(* IEC 61131-3 sources: test/Class/_AccContMain (part 2) *)

        else
          SetMSGNr(dMSGNumber:=ERR_AUTHORITY_EDITUSER);
        end_if;

      else
        SetMSGNr(dMSGNumber:=ERR_USER_NOTEXIST);
      end_if;

    else
      SetMSGNr(dMSGNumber:=ERR_NO_NAME);
    end_if;

  else
    SetMSGNr(dMSGNumber:=ERR_DELUSER);
  end_if;

END_FUNCTION

FUNCTION GLOBAL _AccContMain::ShowUserData
  VAR
    tmpPos    : DINT;
    tmpUser   : t_s_UserV2;  //V2.29, dacpat, updated to new struct
  END_VAR

  tmpPos := -1;

  // Benutzername angegeben
  //-----------------------------------------------------------------------------------------
  if (StrEditUserName.GetLength()) then

      // Position des Benutzers holen
      //-----------------------------------------------------------------------------------------
      tmpPos := SearchUser(pBuffer := UsersBuffer, pUserName:=StrEditUserName.DataBuffer.GetDataPtr(), pUser:=#tmpUser);
      if (tmpPos >= 0) then

        // Benutzerdaten kopieren
        StrEditUserName.WriteDataOff(udLen:=_strlen(#tmpUser.aUsername[0]), udOff:=0, pData:=#tmpUser.aUsername[0]);
        StrEditPasswordOld.WriteDataOff(udLen:=1, udOff:=0, pData:="");
        StrEditPassword.WriteDataOff(udLen:=1, udOff:=0, pData:="");
        StrEditPassword2.WriteDataOff(udLen:=1, udOff:=0, pData:="");
        StrEditInfo.WriteDataOff(udLen:=_strlen(#tmpUser.aUserInfo[0]), udOff:=0, pData:=#tmpUser.aUserInfo[0]);
        ELevel   := tmpUser.usUserLevel;
        ETimeOut := tmpUser.udUserTimeout;

      else

        // Leere Daten kopieren
        StrEditUserName.WriteDataOff(udLen:=1, udOff:=0, pData:="");
        StrEditPasswordOld.WriteDataOff(udLen:=1, udOff:=0, pData:="");
        StrEditPassword.WriteDataOff(udLen:=1, udOff:=0, pData:="");
        StrEditPassword2.WriteDataOff(udLen:=1, udOff:=0, pData:="");
        StrEditInfo.WriteDataOff(udLen:=1, udOff:=0, pData:="");
        ELevel   := 0;
        ETimeOut := 0;

        SetMSGNr(dMSGNumber:=ERR_USER_NOTEXIST);

      end_if;

  else

    SetMSGNr(dMSGNumber:=ERR_NO_NAME);

  end_if;

END_FUNCTION

FUNCTION GLOBAL _AccContMain::ChangePassword
	VAR_INPUT
		bAdmin 	: BOOL;
	END_VAR
	VAR_OUTPUT
		bRet 	: BOOL;
	END_VAR
  VAR
  	tmpUserName   : ARRAY[0..AccessControl_MaxUsernameLength] of CHAR;
    tmpPassword   : ARRAY[0..AccessControl_MaxPasswordLength] of CHAR;
    tmpPWControl  : ARRAY[0..AccessControl_MaxPasswordLength] of CHAR;
    tmpUser       : t_s_UserV2;  //V2.29, dacpat, updated to new struct
    pActUser      : ^t_s_UserV2;  //V2.29, dacpat, updated to new struct
    tmpPos        : DINT;
    tmpPW1Length  : UDINT;
    tmpPW2Length  : UDINT;
  END_VAR

  bRet            := false;
  tmpUserName[0]  := 0;
  tmpPassword[0]  := 0;
  tmpPWControl[0] := 0;
  pActUser        := NIL;
  tmpPos          := 0;

  // Benutzer eingeloggt oder Benutzerverwaltung
  //-----------------------------------------------------------------------------------------
  if ((UserIsLoggedIn = true) | (bAdmin = true)) then

    // Benutzername und Passwörter holen
    if (bAdmin = true) then
      StrEditUserName.GetDataAt(pData:=#tmpUserName[0], udSize:=StrEditUserName.GetLength()+1, udAt:=0);
    else
      StrActUser.GetDataAt(pData:=#tmpUserName[0], udSize:=StrActUser.GetLength()+1, udAt:=0);
    end_if;
    tmpPW1Length := StrEditPassword.GetLength()+1;
    tmpPW2Length := StrEditPassword2.GetLength()+1;
    StrEditPassword.GetDataAt(pData:=#tmpPassword[0], udSize:=tmpPW1Length, udAt:=0);
    StrEditPassword2.GetDataAt(pData:=#tmpPWControl[0], udSize:=tmpPW2Length, udAt:=0);

    // Soll das PW geändert werden?
    //-----------------------------------------------------------------------------------------
    if ((tmpPW1Length > 1) & (tmpPW2Length > 1)) then

      // Geändertes Passwort richtig eingegeben?
      //-----------------------------------------------------------------------------------------
      if (StrCmp(p0:=#tmpPassword[0], x1:=sizeof(tmpPassword[0]), p2:=#tmpPWControl[0], x3:=sizeof(tmpPWControl[0])) = 0) then

        // Position des Benutzers holen
        tmpPos := SearchUser(pBuffer := UsersBuffer, pUserName:= #tmpUserName[0], pUser:=#tmpUser);
        if (tmpPos >= 0) then

          // Benutzerdaten anhand der Position holen und neues Passwort setzen
          //-----------------------------------------------------------------------------------------
          pActUser := getUserToEdit(udPos:=to_udint(tmpPos));
          if (pActUser <> NIL) then

            StrNCpy(p0 := #pActUser^.aUserPassword[0],
                    x1 := sizeof(pActUser^.aUserPassword[0]),
                    p2 := #tmpPassword[0],
                    x3 := sizeof(tmpPassword[0]),
                    ml := AccessControl_MaxPasswordLength);
            if (bAdmin = false) then
              refreshUserFile();
            end_if;
            SetMSGNr(dMSGNumber:=MSG_PWCHANGE_OK);
            bRet := true;

          end_if;

        else

          SetMSGNr(dMSGNumber:=ERR_USER_NOTEXIST);

        end_if;

      else

        SetMSGNr(dMSGNumber:=ERR_WRONG_PWCHANGE);

      end_if;

    else

      // Passwort nicht geändert
      bRet := FALSE;

    end_if;

  end_if;

END_FUNCTION

FUNCTION VIRTUAL GLOBAL _AccContMain::SelectFunction::Write
	VAR_INPUT
		input (EAX) 	: DINT;
	END_VAR
	VAR_OUTPUT
		result (EAX) 	: DINT;
	END_VAR

	SelectFunction := input;

  //*****************************************************************************
  //** Jeweilige Funktion ausgewählt                                           **
  //*****************************************************************************
  case SelectFunction of

    // Legt einen neuen Benutzer an
    1:  AddUser();
        clearServers();

    // Löscht den ausgewählten Benutzer
    2:  DeleteUser();
        clearServers();

    // Bearbeitet den ausgewählten Benutzer
    3:  EditUser();
        clearServers();

    // Login
    4:  Login();
        clearServers();

    // Logout
    5:  Logout();
        clearServers();

    // Schreibt die Benutzerdaten des ausgewählten Benutzers auf die Server zum Bearbeiten
    6:  ShowUserData();

    // Ändert das Passwort des ausgewählten Benutzers
    7:  ChangePassword(bAdmin:=false);
        clearServers();

    // Verknüpft die Seriennummer des aktuellen Speichermediums mit dem eingeloggten Benutzer
    8:  AddUsbSN();
        clearServers();

    // Verknüpft die Seriennummer des aktuellen Speichermediums mit dem eingeloggten Benutzer
    9:  AddUsbSNbyUser();
        clearServers();

    // Löscht die Verknüpfung der Seriennummer mit dem aktuellen Speichermedium
    10: DelUsbSN();
        clearServers();

    // Löscht alle Benutzerdaten auf den Servern
    11: clearServers();

    // Springt auf den vorherigen Bildschirm
    12: closeScreen();

    // V2.30, dacpat, RFID Login
    13:  IsRFIDUser := TRUE;
         Login();
         clearServers();

    // V2.30, dacpat, RFID Add User
    14:  IsRFIDUser := TRUE;
         AddUser();
         clearServers();

  end_case;

 	result := SelectFunction;
  SelectFunction := 0;

END_FUNCTION

FUNCTION _AccContMain::SearchUser
	VAR_INPUT
		pBuffer 	: ^t_s_VKUser;
		pUserName 	: ^USINT;
		pUser   : ^t_s_UserV2;  //V2.29, dacpat, updated to new struct
	END_VAR
	VAR_OUTPUT
		retcode 	: DINT;
	END_VAR
  VAR
  	tmpPos        : DINT;
    pActualVKUser : ^t_s_VKUser;
  END_VAR

  retcode := -1;

  if (pBuffer = NIL) then
    return;
  end_if;;

  tmpPos  := 0;

  pActualVKUser := pBuffer;

  // Benutzer anhand des Benutzernamens suchen
  //-----------------------------------------------------------------------------------------
  while (pActualVKUser <> NIL) do

    tmpPos += 1;
    if (StrCmp(p0:=#pActualVKUser^.User.aUsername[0], x1:=sizeof(pActualVKUser^.User.aUsername[0]), p2:=pUserName, x3:=sizeof(_ASCII)) = 0) then

      // Benutzerdaten zurückgeben
      if (pUser <> NIL) then
        pUser^ := pActualVKUser^.User;
      end_if;

      retcode := tmpPos-1;
      exit;

    else

      pActualVKUser := pActualVKUser^.pNext;
      retcode       := -1;

    end_if;

  end_while;

END_FUNCTION

FUNCTION VIRTUAL GLOBAL _AccContMain::Login
  VAR
    tmpUser       : t_s_UserV2;  //V2.29, dacpat, updated to new struct
    tmpUserName   : ARRAY[0..AccessControl_MaxUsernameLength] of CHAR;
    tmpPassword   : ARRAY[0..AccessControl_MaxPasswordLength] of CHAR;
    tmpScreenInfo : ^_PRJ_ENTRY;
    NiGive	      : CmdStruct;
    NiGet         : Results;
    tmpPos        : DINT;
    pEditUser     : ^t_s_UserV2;  //V2.29, dacpat, updated to new struct
  END_VAR

  tmpUserName[0] := 0;
  tmpPassword[0] := 0;

  // Benutzername und Passwort holen
  StrLoginUserName.GetDataAt(pData:=#tmpUserName[0], udSize:=StrLoginUserName.GetLength()+1, udAt:=0);
  StrLoginPassword.GetDataAt(pData:=#tmpPassword[0], udSize:=StrLoginPassword.GetLength()+1, udAt:=0);

  // Benutzername angegeben?
  //-----------------------------------------------------------------------------------------
  if (StrLoginUserName.GetLength()) then
  (*
    // Administrator holen
    if UsersBuffer = NIL then

      //UsersBuffer$^void := coSystem.Malloc(sizeof(t_s_VKUser));
      //UsersBuffer^.pNext := NIL;
      //tmpUser := UsersBuffer^.User;

    else

      tmpUser := UsersBuffer^.User;

    end_if;
    *)

    _memset(dest:=#tmpUser, usByte:=0, cntr:=sizeof(t_s_UserV2));  //V2.29, dacpat, updated to new struct

    // Wenn der Benutzer existiert oder sich der Administrator einloggt
    //-----------------------------------------------------------------------------------------
    // sprdie v2.24 - save pos of user if normal user logged in
    tmpPos := SearchUser(pBuffer := UsersBuffer, pUserName:=#tmpUserName[0], pUser:=#tmpUser);
    if ( (tmpPos >= 0) |
         (SearchUser(pBuffer := StandardUser, pUserName:=#tmpUserName[0], pUser:=#tmpUser) >= 0) ) then

      // Passwort überprüfen
      if (StrCmp(p0:=#tmpUser.aUserPassword[0], x1:=sizeof(tmpUser.aUserPassword[0]), p2:=#tmpPassword[0], x3:=sizeof(tmpPassword[0])) = 0) then

        // Wenn ein anderer Benutzer eingeloggt ist, diesen ausloggen
        if (UserIsLoggedIn = true) then
          bLogoutOldUser := true;
          Logout();
          bLogoutOldUser := false;
        end_if;

        // Neuen Benutzer einloggen
        StrActUser.WriteDataOff(udLen:=_strlen(#tmpUser.aUsername[0]), udOff:=0, pData:=#tmpUser.aUsername[0]);
        ActLevel       := tmpUser.usUserLevel;
        UserIsLoggedIn := true;

        // Login als Event speichern
        if (IsCon_ccEventQueue = True) then
          NiGive.uiCmd    := 7;               // Command AddUserLoginLogout()
          NiGive.aPara[0] := (#tmpUser.aUsername[0])$DINT;
          NiGive.aPara[1] := ActLevel;
          NiGive.aPara[2] := TO_DINT(TRUE);
          ccEventQueue.NewInst(#NiGive, #NiGet);
        end_if;

        // sprdie v2.24 - save login date & time of user
        if tmpPos >= 0 then
          pEditUser := getUserToEdit(tmpPos$UDINT);
          get_DATIM(#pEditUser^.LastLogin);
        end_if;

        // Zeit beim Login speichern (für Abmeldezeit)
        udTimeout := ops.tAbsolute;

        // Soll Benutzer-Level überprüft werden?
        if (bdAccessConfig.IgnoreScreenAccess = 0) then

          // Neuer Benutzer berechtigt auf diesem Screen zu sein?
          tmpScreenInfo := Prj_GetEntryByNo(x0:=to_uint(ActScreenNr.Read()), x1:=_PE_PICTURE);
          if ((tmpScreenInfo <> NIL) & (tmpScreenInfo^.access > ActLevel)) then
            bCloseScreen := true;
            closeScreen();
            SetMSGNr(dMSGNumber:=ERR_NO_SCREEN_ACCESS);
            IsRFIDUser := FALSE;
            return;
          end_if;

        end_if;

        // Seite refreshen
        IsRFIDUser := FALSE;
        InsertCmd(x0:=CMD_NEWPICTURE, x1:=to_dint(ActScreenNr.Read()), x2:=0);

      else

        IsRFIDUser := FALSE;
        SetMSGNr(dMSGNumber:=ERR_WRONG_PASS);

      end_if;

    else

      //V2.30, dacpat, a new RFID can be added to the user list when the user doesnt exist
      if IsRFIDUser = TRUE then

        // Allow the RFID user to be added to the user list.
        SetMSGNr(dMSGNumber := MSG_RFID_ADDUSER);
      else

        // Normal user handling
        SetMSGNr(dMSGNumber:=ERR_USER_NOTEXIST);
      end_if;
      //SetMSGNr(dMSGNumber:=ERR_USER_NOTEXIST);

    end_if;

  else

    IsRFIDUser := FALSE;
    SetMSGNr(dMSGNumber:=ERR_NO_NAME);

  end_if;

  SaveUsersToRamEx();

END_FUNCTION

FUNCTION VIRTUAL GLOBAL _AccContMain::Logout
  VAR
    tmpUserName   : ARRAY[0..AccessControl_MaxUsernameLength] of CHAR;
    tmpScreenInfo : ^_PRJ_ENTRY;
    NiGive        : CmdStruct;
    NiGet         : Results;
    tmpPos        : DINT;
    pEditUser     : ^t_s_UserV2;  //V2.29, dacpat, updated to new struct
    tmpUser       : t_s_UserV2;  //V2.29, dacpat, updated to new struct
  END_VAR

  // Logout als Event speichern
  //-----------------------------------------------------------------------------------------
  tmpUserName[0] := 0;
  StrActUser.GetDataAt(pData:=#tmpUserName[0], udSize:=StrActUser.GetLength()+1, udAt:=0);
  if (IsCon_ccEventQueue = True) then
    NiGive.uiCmd    := 7;               // Command AddUserLoginLogout()
    NiGive.aPara[0] := (#tmpUserName[0])$DINT;
    NiGive.aPara[1] := ActLevel;
    NiGive.aPara[2] := TO_DINT(FALSE);
    ccEventQueue.NewInst(#NiGive, #NiGet);
  end_if;

  // sprdie v2.24 - save date & time of logout
  tmpPos := SearchUser(pBuffer := UsersBuffer, pUserName:=#tmpUserName[0], pUser:=#tmpUser);
  if tmpPos >= 0 then
    pEditUser := getUserToEdit(tmpPos$UDINT);
    get_DATIM(#pEditUser^.LastLogout);
  end_if;

  // Aktuelle Benutzerdaten zurücksetzen
  //-----------------------------------------------------------------------------------------
  StrActUser.WriteDataOff(udLen:=1, udOff:=0, pData:="");
  ActLevel        := 0;
  UserIsLoggedIn  := false;
  LoggedInWithUsb := false;

  // Soll Benutzer-Level überprüft werden?
  if (bdAccessConfig.IgnoreScreenAccess = 0) then

    // Benutzer berechtigt auf diesem Bildschirm zu sein?
    tmpScreenInfo := Prj_GetEntryByNo(x0:=to_uint(ActScreenNr.Read()), x1:=_PE_PICTURE);
    if ((bLogoutOldUser = false) & (tmpScreenInfo <> NIL) & (tmpScreenInfo^.access > ActLevel)) then
      bCloseScreen := true;
      closeScreen();
      SetMSGNr(dMSGNumber:=ERR_NO_SCREEN_ACCESS);
    end_if;

  end_if;
  RefreshList.Write(input:=1);
  SaveUsersToRamEx();

END_FUNCTION

FUNCTION _AccContMain::clearServers

  // Alle Server zurücksetzen/löschen
  //-----------------------------------------------------------------------------------------
  StrEditPasswordOld.Clear();
  StrEditPassword.Clear();
  StrEditPassword2.Clear();
  StrEditUserName.Clear();
  StrEditInfo.Clear();
  StrLoginPassword.Clear();
  StrLoginUserName.Clear();
  ELevel   := 0;
  ETimeOut := 0;

END_FUNCTION

FUNCTION VIRTUAL GLOBAL _AccContMain::SetMSGNr
	VAR_INPUT
		dMSGNumber 	: DINT;
	END_VAR

  // Info für Pop-Up Fenster in der Visualisierung
  MSGNr := dMSGNumber;
  doWindowOpen := TRUE;

END_FUNCTION

FUNCTION GLOBAL _AccContMain::getUserDataByNr
	VAR_INPUT
		udUserNr 	: UDINT;
		pUser 	: ^t_s_UserV2;  //V2.29, dacpat, updated to new struct
	END_VAR
	VAR_OUTPUT
		retcode 	: DINT;
	END_VAR
  VAR
  	tmpPos        : UDINT;
    pActualVKUser : ^t_s_VKUser;
  END_VAR

  tmpPos  := 0;
  pActualVKUser := UsersBuffer;

  // Übergabeparameter ok?
  //-----------------------------------------------------------------------------------------
  if ((pUser <> NIL) & (udUserNr >= 0)) then

    // Benutzer anhand der Nummer suchen
    //-----------------------------------------------------------------------------------------
    while ((tmpPos <> udUserNr) & (pActualVKUser <> NIL) & (pActualVKUser^.pNext <> NIL)) do

      tmpPos        += 1;
      pActualVKUser := pActualVKUser^.pNext;

    end_while;

    // Gefundene Benutzerdaten gültig?
    //-----------------------------------------------------------------------------------------
    if (pActualVKUser <> NIL) then
      pUser^  := pActualVKUser^.User;
      retcode := 0;
    else
      retcode := -1;
    end_if;

  else

    retcode := -1;

  end_if;

END_FUNCTION

FUNCTION GLOBAL _AccContMain::getNumberOfUsers
	VAR_OUTPUT
		udUsers 	: UDINT;
	END_VAR

  udUsers := udNumberOfUsers;

END_FUNCTION

FUNCTION _AccContMain::getUserToEdit
	VAR_INPUT
		udPos 	: UDINT;
	END_VAR
	VAR_OUTPUT
		pUser 	: ^t_s_UserV2;  //V2.29, dacpat, updated to new struct
	END_VAR
  VAR
  	pActualVKUser : ^t_s_VKUser;
    tmpCount      : UDINT;
  END_VAR

  pActualVKUser := UsersBuffer;
  tmpCount := 0;
  pUser    := NIL;

  // Suche Benutzer anhand der Position
  //-----------------------------------------------------------------------------------------
  while ((pActualVKUser <> NIL) & (tmpCount <> udPos)) do
    tmpCount += 1;
    pActualVKUser := pActualVKUser^.pNext;
  end_while;

  // Benutzerdaten zurückgeben (nicht den Administrator -> pos = 0)
  //-----------------------------------------------------------------------------------------
  if (tmpCount >= 0) then
    pUser := #pActualVKUser^.User;
  end_if;

END_FUNCTION

FUNCTION GLOBAL _AccContMain::RegisterAccessList
	VAR_INPUT
		pNewAccessList 	: ^_AccContList;
	END_VAR
  VAR
  	pHelp  : ^t_s_VKAccessLists;
  END_VAR

  // Registrierte Zugriffsliste für Aktualisierung
  //-----------------------------------------------------------------------------------------
  if (pNewAccessList <> NIL) then

    // Speicher leer
    if (pAccessListsBuffer = NIL) then

      pAccessListsBuffer$^void := coSystem.Malloc(size0:=sizeof(t_s_VKAccessLists));
      if (pAccessListsBuffer = NIL) then
        SetMSGNr(dMSGNumber:=ERR_MEMORY);
        LogMyText("_AccContMain::RegisterAccessList(): Fehler beim allokieren des Speichers" );
        return;
      end_if;
      pAccessListsBuffer^.AccessList := pNewAccessList;
      pAccessListsBuffer^.pNext      := NIL;

    else

      // Das Ende der Liste finden
      pHelp := pAccessListsBuffer;
      while (pHelp^.pNext <> NIL) do
        pHelp := pHelp^.pNext;
      end_while;

      // Speicher für die Zugriffsliste allokieren
      pHelp^.pNext$^void := coSystem.Malloc(size0:=sizeof(t_s_VKAccessLists));
      if (pHelp^.pNext = NIL) then
        SetMSGNr(dMSGNumber:=ERR_MEMORY);
        LogMyText("_AccContMain::RegisterAccessList(): Fehler beim allokieren des Speichers" );
        return;
      end_if;
      pHelp^.pNext^.AccessList := pNewAccessList;
      pHelp^.pNext^.pNext      := NIL;

    end_if;
  end_if;

END_FUNCTION

FUNCTION _AccContMain::_AccContMain
	VAR_OUTPUT
		ret_code 	: ConfStates;
	END_VAR

  // Server
  LoggedInWithUsb     := false;
  UserIsLoggedIn      := false;
  ELevel              := 0;
  ETimeOut            := 0;
  // Variablen
  pAccessListsBuffer  := NIL;
  UsersBuffer  := NIL;
  StandardUser := NIL;
  udNumberOfUsers     := 0;
  dErrorCode          := MSG_NO_ERR;

	ret_code            := C_OK;

END_FUNCTION

FUNCTION GLOBAL _AccContMain::NewStick
	VAR_INPUT
		pSerNum 	: ^void;
	END_VAR
  VAR
  	User : t_s_UserV2;  //V2.29, dacpat, updated to new struct
  END_VAR

  StrEditUsbSN.WriteDataOff(udLen:=_strlen(pSerNum$^CHAR), udOff:=0, pData:=pSerNum$^CHAR);

  // Seriennummer des USB-Sticks mit vorhandenen Benutzerdaten vergleichen
  //-----------------------------------------------------------------------------------------
  if (SearchUserbyUsbSN(#User) >= 0) then

    StrLoginUserName.WriteDataOff(udLen:=_strlen(#User.aUsername[0]), udOff:=0, pData:=#User.aUsername[0]);
    StrLoginPassword.WriteDataOff(udLen:=_strlen(#User.aUserPassword[0]), udOff:=0, pData:=#User.aUserPassword[0]);
    Login();
    clearServers();
    LoggedInWithUsb := true;

  elsif (!!bUsersBufferAllocated) then
    bNewStickAtStart := TRUE;
    aPerSerNum := pSerNum$^t_a_USB_SerialV2^;  //V2.29, dacpat, updated to new struct
  end_if;

END_FUNCTION

FUNCTION GLOBAL _AccContMain::StickRemoved
	VAR_INPUT
		pSerNum 	: ^void;
	END_VAR
  VAR
  	tmpUser     : t_s_UserV2;  //V2.29, dacpat, updated to new struct
    tmpUserName : ARRAY[0..AccessControl_MaxUsernameLength] of CHAR;
  END_VAR

  tmpUserName[0] := 0;

  // Nur wenn ein Benutzer mit dem USB-Stick eingeloggt ist
  //-----------------------------------------------------------------------------------------
  if (LoggedInWithUsb = true) then

    StrActUser.GetDataAt(pData:=#tmpUserName[0], udSize:=StrActUser.GetLength()+1, udAt:=0);

    // Benutzerdaten holen
    if (SearchUser(pBuffer := UsersBuffer, pUserName:=#tmpUserName[0], pUser:=#tmpUser) >= 0) then

      // Wenn die Seriennummer identisch ist
      if (StrCmp(p0:=#tmpUser.USBSerial[0], x1:=sizeof(tmpUser.USBSerial[0]), p2:=pSerNum$^CHAR, x3:=sizeof(_ASCII)) = 0) then

        Logout();
        clearServers();
        LoggedInWithUsb := false;

      end_if;

    end_if;

  end_if;

  StrEditUsbSN.Clear();

END_FUNCTION

FUNCTION _AccContMain::SearchUserbyUsbSN
	VAR_INPUT
		pUser 	: ^t_s_UserV2;  //V2.29, dacpat, updated to new struct
	END_VAR
	VAR_OUTPUT
		retcode 	: DINT;
	END_VAR
  VAR
  	tmpPos        : DINT;
    pActualVKUser : ^t_s_VKUser;
    tmpEditUsbSN  : Array[0..AccessControl_MaxUSBSNLengthV2] of CHAR;  //V2.29, dacpat, extended serial number length
  END_VAR

  retcode         := -1;
  tmpPos          := 0;
  tmpEditUsbSN[0] := 0;
  pActualVKUser   := UsersBuffer;

  if (pActualVKUser = NIL) then
    return;
  end_if;

  if (StrEditUsbSN.GetLength() + 1) <= sizeof(tmpEditUsbSN) then  //V2.29, dacpat, check if the data fits into the array or not

    StrEditUsbSN.GetDataAt(pData:=#tmpEditUsbSN[0], udSize:=(StrEditUsbSN.GetLength() + 1), udAt:=0);
  else

    return;
  end_if;

  // Nach der Seriennummer suchen
  //-----------------------------------------------------------------------------------------
  while pActualVKUser <> NIL do

    tmpPos += 1;
    // Gleiche Seriennummer gefunden
    if (StrCmp(p0:=#pActualVKUser^.User.USBSerial[0], x1:=sizeof(pActualVKUser^.User.USBSerial[0]), p2:=#tmpEditUsbSN[0], x3:=sizeof(tmpEditUsbSN[0])) = 0) then

      // Benutzerdaten holen
      if (pUser <> NIL) then
        pUser^ := pActualVKUser^.User;
      end_if;

      retcode := tmpPos-1;
      exit;

    else

      pActualVKUser := pActualVKUser^.pNext;
      retcode := -1;

    end_if;

  end_while;

END_FUNCTION

FUNCTION GLOBAL _AccContMain::AddUsbSNbyUser
  VAR
    tmpUserName : ARRAY[0..AccessControl_MaxUsernameLength] of CHAR;
  END_VAR

  tmpUserName[0] := 0;

  // Eingeloggten Benutzer mit der Seriennummer des USB-Sticks verknüpfen
  //-----------------------------------------------------------------------------------------
  if (UserIsLoggedIn = true) then

    StrActUser.GetDataAt(pData:=#tmpUserName[0], udSize:=StrActUser.GetLength()+1, udAt:=0);
    StrEditUserName.WriteDataOff(udLen:=_strlen(#tmpUserName[0]), udOff:=0, pData:=#tmpUserName[0]);
    AddUsbSN();

  end_if;

END_FUNCTION

FUNCTION GLOBAL _AccContMain::AddUsbSN
  VAR
    tmpPos      : DINT;
    pActUser    : ^t_s_UserV2;  //V2.29, dacpat, updated to new struct
    pOldUserSN      : ^t_s_UserV2;  //V2.29, dacpat, updated to new struct
    tmpUserName     : ARRAY[0..AccessControl_MaxUsernameLength] of CHAR;
    tmpActUserName  : ARRAY[0..AccessControl_MaxUsernameLength] of CHAR;
    tmpNewPos       : DINT;
    tmpOwnUser      : UINT;
  END_VAR

  if UserIsLoggedIn then
    StrActUser.GetDataAt(pData:=#tmpActUserName[0], udSize:=StrActUser.GetLength()+1, udAt:=0);
  end_if;

  tmpPos          := 0;
  pActUser        := NIL;
  tmpUserName[0]  := 0;
  tmpNewPos       := 0;

  // Benutzername angegeben
  //-----------------------------------------------------------------------------------------
  if (StrEditUserName.GetLength()) then

    // Benutzername und dessen Position holen
    StrEditUserName.GetDataAt(pData:=#tmpUserName[0], udSize:=StrEditUserName.GetLength()+1, udAt:=0);
    tmpNewPos := SearchUser(pBuffer := UsersBuffer, pUserName:= #tmpUserName[0], pUser:=NIL);

    // Benutzer gefunden
    //-----------------------------------------------------------------------------------------
    if (tmpNewPos >= 0) then

      // Wenn ein USB-Stick mit einem Benutzer verknüpft werden soll, muss der Benutzer manuell eingeloggt sein
      if ((LoggedInWithUsb = false) & (StrEditUsbSN.GetLength() > 0)) then

        //Benutzerdaten anhand der Position holen
        pActUser := getUserToEdit(udPos:=to_udint(tmpNewPos));
        tmpOwnUser := (StrCmp(p0:=#pActUser^.aUsername[0], x1:=sizeof(pActUser^.aUsername[0]), p2:=#tmpActUserName[0], x3:=sizeof(tmpActUserName[0])));
        if (pActUser <> NIL) & ((pActUser^.usUserLevel < ActLevel) | (tmpOwnUser = 0)) then

          // Wenn dieser USB-Stick schon mit einem anderen Benutzer verknüpft ist, lösche diese Verbindung
          tmpPos := SearchUserbyUsbSN(pUser:=NIL);
          if (tmpPos >= 0) then
            // Benutzerdaten anhand der Position holen
            pOldUserSN := getUserToEdit(udPos:=to_udint(tmpPos));
            if (StrCmp(p0:=#pActUser^.USBSerial[0], x1:=sizeof(pActUser^.USBSerial[0]), p2:=#pOldUserSN^.USBSerial[0], x3:=sizeof(pOldUserSN^.USBSerial[0])) <> 0) then

              if (pOldUserSN <> NIL) & ((pOldUserSN^.usUserLevel < ActLevel) | (StrCmp(p0:=#pOldUserSN^.aUsername[0], x1:=sizeof(pOldUserSN^.aUsername[0]), p2:=#tmpActUserName[0], x3:=sizeof(tmpActUserName[0])) = 0)) then
                pOldUserSN^.USBSerial[0] := 0;
              else
                SetMSGNr(dMSGNumber:=ERR_AUTHORITY_EDITUSER);
                return;
              end_if;

            else
              SetMSGNr(dMSGNumber:=ERR_USB_SERNUM);
            end_if;

          end_if;

          // Seriennummer des USB-Sticks speichern
          StrEditUsbSN.GetDataAt(pData:=#pActUser^.USBSerial[0], udSize:=StrEditUsbSN.GetLength()+1, udAt:=0);
          refreshUserFile();

        else

          SetMSGNr(dMSGNumber:=ERR_AUTHORITY_EDITUSER);

        end_if;
      else

        SetMSGNr(dMSGNumber:=ERR_USB_SERNUM);

      end_if;

    else

      SetMSGNr(dMSGNumber:=ERR_USER_NOTEXIST);

    end_if;

  else

    SetMSGNr(dMSGNumber:=ERR_NO_NAME);

  end_if;

END_FUNCTION

FUNCTION VIRTUAL GLOBAL _AccContMain::IF_WindowEnd
	VAR_INPUT
		whoami 	: ^_WHOAMI;
		pic 	: ^void;
	END_VAR

  // Alle Server beim Schließen eines Fensters zurücksetzen
  //-----------------------------------------------------------------------------------------
  if (whoami^.ima <> IMA_TOUCHEDITOR) then

    clearServers();

  end_if;

END_FUNCTION

FUNCTION GLOBAL _AccContMain::DelUsbSN
  VAR
    tmpPos         : DINT;
    tmpOwnUser     : UINT;
    pActUser       : ^t_s_UserV2;  //V2.29, dacpat, updated to new struct
    tmpUserName    : ARRAY[0..AccessControl_MaxUsernameLength] of CHAR;
    tmpActUserName : ARRAY[0..AccessControl_MaxUsernameLength] of CHAR;
  END_VAR

  tmpPos            := 0;
  pActUser          := NIL;
  tmpUserName[0]    := 0;
  tmpActUserName[0] := 0;

  // Benutzername angegeben
  //-----------------------------------------------------------------------------------------
  if (StrEditUserName.GetLength()) then

    StrEditUserName.GetDataAt(pData:=#tmpUserName[0], udSize:=StrEditUserName.GetLength()+1, udAt:=0);
    StrActUser.GetDataAt(pData:=#tmpActUserName[0], udSize:=StrActUser.GetLength()+1, udAt:=0);

    // Position des Benutzers holen
    tmpPos := SearchUser(pBuffer := UsersBuffer, pUserName:=#tmpUserName[0], pUser:=NIL);
    if (tmpPos >= 0) then

      // Benutzerdaten anhand der Position holen
      pActUser := getUserToEdit(to_udint(tmpPos));
      tmpOwnUser := (StrCmp(p0:=#tmpUserName[0], x1:=sizeof(tmpUserName[0]), p2:=#tmpActUserName[0], x3:=sizeof(tmpActUserName[0])));
      if ( (pActUser <> NIL) & ((tmpOwnUser) | ((tmpOwnUser = 0) & (LoggedInWithUsb = 0))) &
         (StrLen(txt:=#pActUser^.USBSerial[0], size:=sizeof(pActUser^.USBSerial[0])) <> 0) ) then

        // Berechtigt um diesen Benutzer zu bearbeiten bzw. den eigenen Benutzer bearbeiten
        if ((pActUser^.usUserLevel < ActLevel) | (tmpOwnUser = 0)) then
          pActUser^.USBSerial[0] := 0;
          refreshUserFile();
        else
          SetMSGNr(dMSGNumber:=ERR_AUTHORITY_EDITUSER);
        end_if;

      else

        SetMSGNr(dMSGNumber:=ERR_DEL_USB_SERNUM);

      end_if;

    else

      SetMSGNr(dMSGNumber:=ERR_USER_NOTEXIST);

    end_if;

  else

    SetMSGNr(dMSGNumber:=ERR_NO_NAME);

  end_if;

END_FUNCTION

FUNCTION VIRTUAL GLOBAL _AccContMain::CopyUserFile::Write
	VAR_INPUT
		input (EAX) 	: DINT;
	END_VAR
	VAR_OUTPUT
		result (EAX) 	: DINT;
	END_VAR

	CopyUserFile := input;

  // Exportieren/Importieren der Benutzerdatei auf einen USB-Speicher
  //-----------------------------------------------------------------------------------------
  if (CopyUserFile <> 0) then

    // USB-Speichermedium auch angeschlossen?
    //-----------------------------------------------------------------------------------------
    if (IsCon_coDriveLetter = TRUE) then          // KaiAnd, V.2.22

      //if ( (coDriveLetter.GetLength() > 0) &
      //     (StrEditUsbSN.GetLength() > 0) ) then  // KaiAnd, V.2.22

      if (coDriveLetter.GetLength() > 0) then  // V2.31: without check of UsbSerialNumber

        //V2.29, dacpat, reworked write method, file copying etc. is now done in bg task
        if (eUserFileState = AccessControl_IDLE) then

          if (CopyUserFile > 0) then
            // V2.29, dacpat, export with new file name
            eUserFileState := AccessControl_EXPORTUSERS;
          else
            // V2.29, dacpat, check version in file header before importing the file
            CheckHeader    := TRUE;
            eUserFileState := AccessControl_FILEOPENV2;
          end_if;
        end_if;

      else  // coDriveLetter with empty string
        CopyUserFile := 0;
        SetMSGNr(dMSGNumber:=ERR_NO_DRIVE);
      end_if;

    else  // coDriveLetter client not connected
      CopyUserFile := 0;
      SetMSGNr(dMSGNumber:=ERR_NO_DRIVE);
    end_if;

  end_if;

  result := CopyUserFile;

END_FUNCTION

FUNCTION _AccContMain::closeScreen

  // Benutzer befindet sich auf einem Screen, ohne korrekte Zugangsberechtigung
  if ((bCloseScreen = true) & (bdAccessConfig.IgnoreScreenAccess = 0)) then

    // Kehre zum Start-Bildschirm zurück
    InsertCmd(x0:=CMD_NEWPICTURE, x1:=coGlobal.GetStartPicture(), x2:=0);
    bCloseScreen := false;

  end_if;

END_FUNCTION

FUNCTION GLOBAL _AccContMain::CreateAdmin
	VAR_INPUT
		pUsername 	: ^CHAR;
		pPassword 	: ^CHAR;
		usLevel 	: USINT;
	END_VAR
	VAR_OUTPUT
		bSuccessful 	: BOOL;
	END_VAR

  //Rückgabewert initialisieren
  bSuccessful := FALSE;

  if (StandardUser = NIL) then

    StandardUser$^void := coSystem.Malloc(sizeof(t_s_VKUser));
    StandardUser^.pNext := NIL;

  end_if;

  //Benutzerdaten gültig?
  if ((pUsername <> NIL) & (pPassword <> NIL) & (usLevel <> NIL)) then

    StrNCpy(p0 := #StandardUser^.User.aUsername[0],
            x1 := sizeof(StandardUser^.User.aUsername[0]),
            p2 := pUsername,
            x3 := sizeof(_ASCII),
            ml := AccessControl_MaxUsernameLength);
    StrNCpy(p0 := #StandardUser^.User.aUserPassword[0],
            x1 := sizeof(StandardUser^.User.aUserPassword[0]),
            p2 := pPassword,
            x3 := sizeof(_ASCII),
            ml := AccessControl_MaxPasswordLength);
    StandardUser^.User.usUserLevel   := usLevel;
    StandardUser^.User.udUserTimeout := 0;

    bSuccessful := true;

    // HerMor V.2.27: Set Flag true
    setTmpAdmin(true);
  end_if;

END_FUNCTION

FUNCTION VIRTUAL GLOBAL _AccContMain::IF_ChkEnable
	VAR_INPUT
		key 	: DINT;
	END_VAR
	VAR_OUTPUT
		retcode 	: BOOL;
	END_VAR

  retcode := false;

  // Zugangsebenen deaktiviert (frei zugänglich)
  //-----------------------------------------------------------------------------------------
  if (Deactivate = true) then

    retcode := true;

  // Zugangsebenen über NewInst() deaktiviert (frei zugänglich)
  //-----------------------------------------------------------------------------------------
  elsif (bCheckAccesslevel = TRUE) then

    retcode := true;

  // Zugangscode prüfen
  //-----------------------------------------------------------------------------------------
  elsif (ActLevel >= key) then

    retcode := true;

  end_if;

END_FUNCTION

FUNCTION _AccContMain::LogMyText
  VAR_INPUT
		pLogTxt 	: ^CHAR;
	END_VAR

  VAR
    NiGive	  : CmdStruct;
    NiGet     : Results;
  END_VAR

  if ((IsCon_ccSystemLogging = True) & (pLogTxt <> NIL)) then

    NiGive.uiCmd    := 0;               // Command
    NiGive.aPara[0] := (pLogTxt)$DINT;  // pointer to text

    ccSystemLogging.NewInst(#NiGive, #NiGet);

  end_if;

END_FUNCTION

FUNCTION _AccContMain::DeactiveAccessLevel
	VAR_INPUT
		bCheckAccessState 	: DINT;
	END_VAR
	VAR_OUTPUT
		ret_code 	: IprStates;
	END_VAR

  // SchDom V 2.23: Deacivate check accesslevel
  if (bCheckAccessState = TRUE) then
    bCheckAccesslevel := TRUE;
  else
    bCheckAccesslevel := FALSE;
  end_if;

	ret_code := READY;

END_FUNCTION

FUNCTION _AccContMain::SaveUsersToRamEx
  VAR
    i     : UINT;
    pRead : ^t_s_UserV2;  //V2.29, dacpat, updated to new struct
  END_VAR

  ExtUserData.SetSize(udSize:=sizeof(t_s_UserV2)*udNumberOfUsers);  //V2.29, dacpat, updated to new struct

  // loop through users and save to SRAM
  i := 0;
  repeat

    pRead := getUserToEdit(udPos:=i);

    if pRead <> NIL then
      ExtUserData.SetDataAt(pData:=pRead$^USINT, udSize:=sizeof(t_s_UserV2), udAt:=i*sizeof(t_s_UserV2));  //V2.29, dacpat, updated to new struct
    end_if;

    i += 1;

  until (pRead = NIL) end_repeat;

END_FUNCTION

FUNCTION _AccContMain::GetLogTimesFromRamEx
  VAR
    pReadV1      : ^t_s_User;
    pReadV2      : ^t_s_UserV2;  //V2.29, dacpat, updated to new struct
    pWrite       : ^t_s_UserV2;  //V2.29, dacpat, updated to new struct
    dWriteIndex  : DINT;
    noUsers      : UINT;
    i            : UINT;
  END_VAR

  if IsV1 = TRUE & LoadRamExV2 = FALSE then  //V2.29, dacpat, check if version 1 should be used

    pReadV1$^USINT := ExtUserData.GetDataPtr(); // for reading purposes only!!!
    noUsers := to_uint(ExtUserData.m_udLength / sizeof(t_s_User));

    if (pReadV1 <> NIL) & (noUsers > 0) then
      for i:=0 to (noUsers-1) do

        dWriteIndex := SearchUser(pBuffer:=UsersBuffer, pUserName:=#pReadV1^.aUsername[0], pUser:=NIL);

        if dWriteIndex >= 0 then
          pWrite := getUserToEdit(to_udint(dWriteIndex));
          if pWrite <> NIL then
            pWrite^.LastLogin  := pReadV1^.LastLogin;
            pWrite^.LastLogout := pReadV1^.LastLogout;
          end_if;
        end_if;

        pReadV1 += sizeof(t_s_User);
      end_for;

      // Save the users to RamEx in the new format after reading the old format
      SaveUsersToRamEx();
    end_if;
  else

    pReadV2$^USINT := ExtUserData.GetDataPtr(); // for reading purposes only!!!
    noUsers := to_uint(ExtUserData.m_udLength / sizeof(t_s_UserV2));

    if (pReadV2 <> NIL) & (noUsers > 0) then
      for i:=0 to (noUsers-1) do

        dWriteIndex := SearchUser(pBuffer:=UsersBuffer, pUserName:=#pReadV2^.aUsername[0], pUser:=NIL);

        if dWriteIndex >= 0 then
          pWrite := getUserToEdit(to_udint(dWriteIndex));
          if pWrite <> NIL then
            pWrite^.LastLogin  := pReadV2^.LastLogin;
            pWrite^.LastLogout := pReadV2^.LastLogout;
          end_if;
        end_if;

        pReadV2 += sizeof(t_s_UserV2);
      end_for;

      LoadRamExV2.Write(input := FALSE);
    end_if;
  end_if;

END_FUNCTION

// HerMor V2.27:
FUNCTION GLOBAL _AccContMain::getTmpAdmin
	VAR_OUTPUT
		bTmpAdmin 	: BOOL;
	END_VAR

  bTmpAdmin := bCheckTempAdmin;

END_FUNCTION

// HerMor V2.27:
FUNCTION GLOBAL _AccContMain::setTmpAdmin
	VAR_INPUT
		bTmpAdmin 	: BOOL;
	END_VAR

  bCheckTempAdmin := bTmpAdmin;

END_FUNCTION

// HerMor V.2.28:
FUNCTION VIRTUAL GLOBAL _AccContMain::IF_OpenTouchEditor
	VAR_INPUT
		pe 	: ^_EDITOR;
		preselect 	: UINT;
	END_VAR
	VAR_OUTPUT
		retcode 	: UINT;
	END_VAR

  VAR
  	CheckASCII : BDINT;
  END_VAR

  CheckASCII := Config.Read();

  //Überprüfen, ob Config-Bit0 gesetzt ist (NUR SETZTEN WENN FILEEXPLORER IMPLEMENTIERT IST!!)
  if (CheckASCII AND 2#1) then
    // Tastatur wird geändert wenn nur ASCII Zeichen erlaubt sind
    if (VarList_GetOnlyAscii(x0 := #pe^.variable.info) = TRUE) then
      // Eingabe nur ASCII
      if (preselect = _WIN_EDITOR_ANUMERIC) then
        // ASCII Tastatur aufrufen
        preselect := _WIN_EDITOR_ANUMFILEX;
      end_if;
    end_if;
  end_if;

  retcode := preselect;

END_FUNCTION

FUNCTION _AccContMain::ConvertV1UserData
	VAR_INPUT
		pUserDataV1 	: ^t_s_User;
		pUserDataV2 	: ^t_s_UserV2;
	END_VAR

  //V2.29, dacpat, convert the old user data into the new format

  // User name
  //-----------------------------------------------------------------------------------------
  StrNCpy(p0 := #pUserDataV2^.aUsername[0],
          x1 := sizeof(pUserDataV2^.aUsername[0]),
          p2 := #pUserDataV1^.aUsername[0],
          x3 := sizeof(_ASCII),
          ml := AccessControl_MaxUsernameLength);

  // User password
  //-----------------------------------------------------------------------------------------
  StrNCpy(p0 := #pUserDataV2^.aUserPassword[0],
          x1 := sizeof(pUserDataV2^.aUserPassword[0]),
          p2 := #pUserDataV1^.aUserPassword[0],
          x3 := sizeof(_ASCII),
          ml := AccessControl_MaxPasswordLength);

  // User level
  //-----------------------------------------------------------------------------------------
  pUserDataV2^.usUserLevel := pUserDataV1^.usUserLevel;

  // User timeout
  //-----------------------------------------------------------------------------------------
  pUserDataV2^.udUserTimeout := pUserDataV1^.udUserTimeout;

  // User info
  //-----------------------------------------------------------------------------------------
  StrNCpy(p0 := #pUserDataV2^.aUserInfo[0],
          x1 := sizeof(pUserDataV2^.aUserInfo[0]),
          p2 := #pUserDataV1^.aUserInfo[0],
          x3 := sizeof(_ASCII),
          ml := AccessControl_MaxUserInfoLength);

  // User serial number
  //-----------------------------------------------------------------------------------------
  StrNCpy(p0 := #pUserDataV2^.USBSerial[0],
          x1 := sizeof(pUserDataV2^.USBSerial[0]),
          p2 := #pUserDataV1^.USBSerial[0],
          x3 := sizeof(_ASCII),
          ml := AccessControl_MaxUSBSNLength);

  // User last login
  //-----------------------------------------------------------------------------------------
  pUserDataV2^.LastLogin := pUserDataV1^.LastLogin;

  // User last logout
  //-----------------------------------------------------------------------------------------
  pUserDataV2^.LastLogout := pUserDataV1^.LastLogout;

END_FUNCTION

FUNCTION GLOBAL _AccContMain::SetRFIDMsgNr
	VAR_INPUT
		dMSGNumber 	: DINT;
	END_VAR

  //V2.30, dacpat, new method to open the new window for special RFID messages

  IsRFIDUser := TRUE;  // Set flag to open different message window
  SetMSGNr(dMSGNumber := dMSGNumber);

END_FUNCTION

FUNCTION GLOBAL _AccContMain::GetActUser
  VAR_INPUT
		pUser 	: ^CHAR;
	END_VAR
  VAR
  	tmpUser : ARRAY [0..AccessControl_MaxUsernameLength] of CHAR;
    tmpSize : UDINT;
  END_VAR

  //V2.30, dacpat, new method to get usernam of the currently logged in  user

  tmpSize := StrActUser.GetLength();

  if tmpSize > AccessControl_MaxUsernameLength then

    tmpSize := AccessControl_MaxUsernameLength;
  end_if;

  StrActUser.GetDataAt(pData  := #tmpUser[0],
                       udSize := tmpSize,
                       udAt   := 0);

  tmpUser[tmpSize] := 0;

  // Copy the ActUser to the given pointer
  StrNCpy(p0 := pUser,
          x1 := sizeof(_ASCII),
          p2 := #tmpUser[0],
          x3 := sizeof(_ASCII),
          ml := AccessControl_MaxUsernameLength);

END_FUNCTION

FUNCTION GLOBAL _AccContMain::SetUserDataStrings
	VAR_INPUT
		StringSelection 	: t_e_UserDataStrings;
		pString 	: ^CHAR;
		StringLength 	: UDINT;
	END_VAR
	VAR_OUTPUT
		Retcode 	: UDINT;
	END_VAR
  VAR
  	tmpSize : UDINT;
  END_VAR

  //V2.30, dacpat, new method to be able to set the different embedde strings from another class

  Retcode := 0;

  if pString <> NIL then

    case StringSelection of

      // StrEditUserName
      //-----------------------------------------------------------------------------------------
      UserData_StrEditUserName:
        // Check the string size
        if StringLength > AccessControl_MaxUsernameLength then

          tmpSize := AccessControl_MaxUsernameLength;
        else

          tmpSize := StringLength;
        end_if;

        StrEditUserName.WriteDataOff(udLen := tmpSize,
                                     udOff := 0,
                                     pData := pString);

      // StrEditPasswordOld
      //-----------------------------------------------------------------------------------------
      UserData_StrEditPasswordOld:
        // Check the string size
        if StringLength > AccessControl_MaxPasswordLength then

          tmpSize := AccessControl_MaxPasswordLength;
        else

          tmpSize := StringLength;
        end_if;

        StrEditPasswordOld.WriteDataOff(udLen := tmpSize,
                                        udOff := 0,
                                        pData := pString);

      // StrEditPassword
      //-----------------------------------------------------------------------------------------
      UserData_StrEditPassword:
        // Check the string size
        if StringLength > AccessControl_MaxPasswordLength then

          tmpSize := AccessControl_MaxPasswordLength;
        else

          tmpSize := StringLength;
        end_if;

        StrEditPassword.WriteDataOff(udLen := tmpSize,
                                     udOff := 0,
                                     pData := pString);

      // StrEditPassword2
      //-----------------------------------------------------------------------------------------
      UserData_StrEditPassword2:
        // Check the string size
        if StringLength > AccessControl_MaxPasswordLength then

          tmpSize := AccessControl_MaxPasswordLength;
        else

          tmpSize := StringLength;
        end_if;

        StrEditPassword2.WriteDataOff(udLen := tmpSize,
                                      udOff := 0,
                                      pData := pString);

      // StrEditInfo
      //-----------------------------------------------------------------------------------------
      UserData_StrEditInfo:
        // Check the string size
        if StringLength > AccessControl_MaxUserInfoLength then

          tmpSize := AccessControl_MaxUserInfoLength;
        else

          tmpSize := StringLength;
        end_if;

        StrEditInfo.WriteDataOff(udLen := tmpSize,
                                 udOff := 0,
                                 pData := pString);

      // StrLoginUserName
      //-----------------------------------------------------------------------------------------
      UserData_StrLoginUserName:
        // Check the string size
        if StringLength > AccessControl_MaxUsernameLength then

          tmpSize := AccessControl_MaxUsernameLength;
        else

          tmpSize := StringLength;
        end_if;

        StrLoginUserName.WriteDataOff(udLen := tmpSize,
                                      udOff := 0,
                                      pData := pString);

      // StrLoginPassword
      //-----------------------------------------------------------------------------------------
      UserData_StrLoginPassword:
        // Check the string size
        if StringLength > AccessControl_MaxPasswordLength then

          tmpSize := AccessControl_MaxPasswordLength;
        else

          tmpSize := StringLength;
        end_if;

        StrLoginPassword.WriteDataOff(udLen := tmpSize,
                                      udOff := 0,
                                      pData := pString);

      else

        Retcode := DEFSCOPE;
        LogMyText("_AccContMain::SetUserDataStrings(): Invalid string selection");
    end_case;
  else

    Retcode := DEFSCOPE;
    LogMyText("_AccContMain::SetUserDataStrings(): Invalid string pointer");
  end_if;

END_FUNCTION

FUNCTION GLOBAL _AccContMain::getUserDataByUser
	VAR_INPUT
		pActUser 	: ^CHAR;
		pUser 	: ^t_s_UserV2;
	END_VAR
	VAR_OUTPUT
		retcode 	: DINT;
	END_VAR
  VAR
  	tmpPos : DINT;
  END_VAR

  //V2.30, dacpat, new method to get the user informations by using the username

  retcode := FALSE;

  if pActUser <> NIL & pUser <> NIL then

    tmpPos := SearchUser(pBuffer   := UsersBuffer,
                         pUserName := pActUser,
                         pUser     := pUser);

    if tmpPos >= 0 then

      // User was found
      retcode := TRUE;
    else

      // User is not in the buffer
      LogMyText("_AccContMain::getUserDataByUser(): User was not found in the buffer");
    end_if;
  else

    LogMyText("_AccContMain::getUserDataByUser(): Invalid pointer");
  end_if;

END_FUNCTION
